FUNCTION_BLOCK "Sequencer"
{ S7_Optimized_Access := 'FALSE' }
VERSION : 0.1
   VAR_OUTPUT
      Dev1 : Bool;
      Dev2 : Bool;
      Dev3 : Bool;
      Dev4 : Bool;
      Dev5 : Bool;
      Dev6 : Bool;
      Dev7 : Bool;
      Dev8 : Bool;
      Dev9 : Bool;
      Dev10 : Bool;
      Dev11 : Bool;
      Dev12 : Bool;
      Dev13 : Bool;
      Dev14 : Bool;
      Dev15 : Bool;
      Dev16 : Bool;
      CurTime : Time;
   END_VAR

   VAR
      Enable : Bool;
      Hold : Bool;
      Seq : "Sequence";
      RstStep { S7_SetPoint := 'True'} : Bool := TRUE;
      Step : Int := "MIN_STEP_NUMB";
      Timer_IN { ExternalAccessible := 'False'; ExternalVisible := 'False'; ExternalWritable := 'False'} : Bool;
      Done : Bool;
      tmr : "TON_200ms";
   END_VAR

   VAR_TEMP
      tAddStep : Bool;
   END_VAR


BEGIN
	// Управление 16-ю механизмами в зависимости
	// от заданной последовательности Seq

	IF #RstStep THEN
	    #Step := "MIN_STEP_NUMB";
	    #Timer_IN := FALSE;
	    #Done := FALSE;
	    #RstStep := FALSE;
	END_IF;

	#tmr(In := #Timer_IN,
	     PT := "intToTime_1"(intTime := #Seq.delay[#Step], select := 0));

	#Timer_IN := #Enable AND (NOT (#tmr.Q OR #Hold OR #Done));
	#CurTime := #tmr.PT - #tmr.ET;

	//Переход к след. шагу
	IF #tmr.Q AND (NOT #Hold) AND (NOT #Done) THEN
	    #Step += 1;
	END_IF;

	IF #Enable THEN //Пропуск шагов с нулевой задержкой
	    WHILE #Seq.delay[#Step] <= 0 DO
	        IF #Step >= "MAX_STEP_NUMB" THEN
	            EXIT;
	        END_IF;
	       #Step += 1;
	    END_WHILE;
	END_IF;


	//Конец последовательности
	IF #Step >= "MAX_STEP_NUMB" THEN
	    #Done := #Enable;
	    RETURN;
	END_IF;

	IF #Enable THEN
	    #Dev1 := #Seq.devOn[#Step, 1];
	    #Dev2 := #Seq.devOn[#Step, 2];
	    #Dev3 := #Seq.devOn[#Step, 3];
	    #Dev4 := #Seq.devOn[#Step, 4];
	    #Dev5 := #Seq.devOn[#Step, 5];
	    #Dev6 := #Seq.devOn[#Step, 6];
	    #Dev7 := #Seq.devOn[#Step, 7];
	    #Dev8 := #Seq.devOn[#Step, 8];
	    #Dev9 := #Seq.devOn[#Step, 9];
	    #Dev10 := #Seq.devOn[#Step, 10];
	    #Dev11 := #Seq.devOn[#Step, 11];
	    #Dev12 := #Seq.devOn[#Step, 12];
	    #Dev13 := #Seq.devOn[#Step, 13];
	    #Dev14 := #Seq.devOn[#Step, 14];
	    #Dev15 := #Seq.devOn[#Step, 15];
	    #Dev16 := #Seq.devOn[#Step, 16];
	END_IF;




END_FUNCTION_BLOCK

